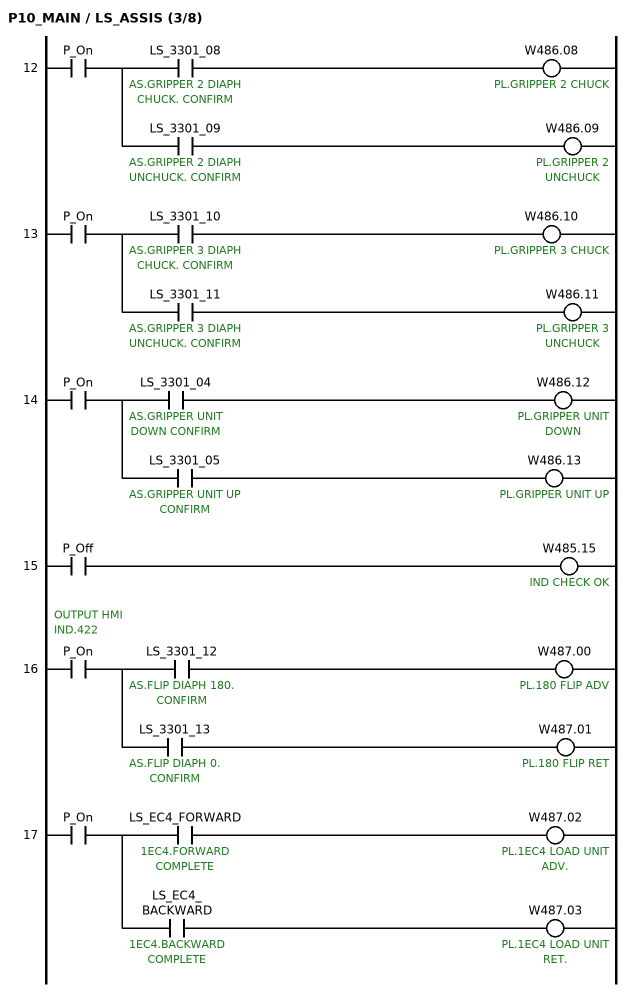
; [picture p48: P10_MAIN / LS_ASSIS, rungs 12-17]
; rung 12
LD P_On
OUT TR0
AND LS_3301_08  ; AS.GRIPPER 2 DIAPH CHUCK. CONFIRM
OUT W486.08  ; PL.GRIPPER 2 CHUCK
LD TR0
AND LS_3301_09  ; AS.GRIPPER 2 DIAPH UNCHUCK. CONFIRM
OUT W486.09  ; PL.GRIPPER 2 UNCHUCK
; rung 13
LD P_On
OUT TR0
AND LS_3301_10  ; AS.GRIPPER 3 DIAPH CHUCK. CONFIRM
OUT W486.10  ; PL.GRIPPER 3 CHUCK
LD TR0
AND LS_3301_11  ; AS.GRIPPER 3 DIAPH UNCHUCK. CONFIRM
OUT W486.11  ; PL.GRIPPER 3 UNCHUCK
; rung 14
LD P_On
OUT TR0
AND LS_3301_04  ; AS.GRIPPER UNIT DOWN CONFIRM
OUT W486.12  ; PL.GRIPPER UNIT DOWN
LD TR0
AND LS_3301_05  ; AS.GRIPPER UNIT UP CONFIRM
OUT W486.13  ; PL.GRIPPER UNIT UP
; rung 15
LD P_Off
OUT W485.15  ; IND CHECK OK
; rung 16: OUTPUT HMI / IND.422
LD P_On
OUT TR0
AND LS_3301_12  ; AS.FLIP DIAPH 180. CONFIRM
OUT W487.00  ; PL.180 FLIP ADV
LD TR0
AND LS_3301_13  ; AS.FLIP DIAPH 0. CONFIRM
OUT W487.01  ; PL.180 FLIP RET
; rung 17
LD P_On
OUT TR0
AND LS_EC4_FORWARD  ; 1EC4.FORWARD COMPLETE
OUT W487.02  ; PL.1EC4 LOAD UNIT ADV.
LD TR0
AND LS_EC4_BACKWARD  ; 1EC4.BACKWARD COMPLETE
OUT W487.03  ; PL.1EC4 LOAD UNIT RET.

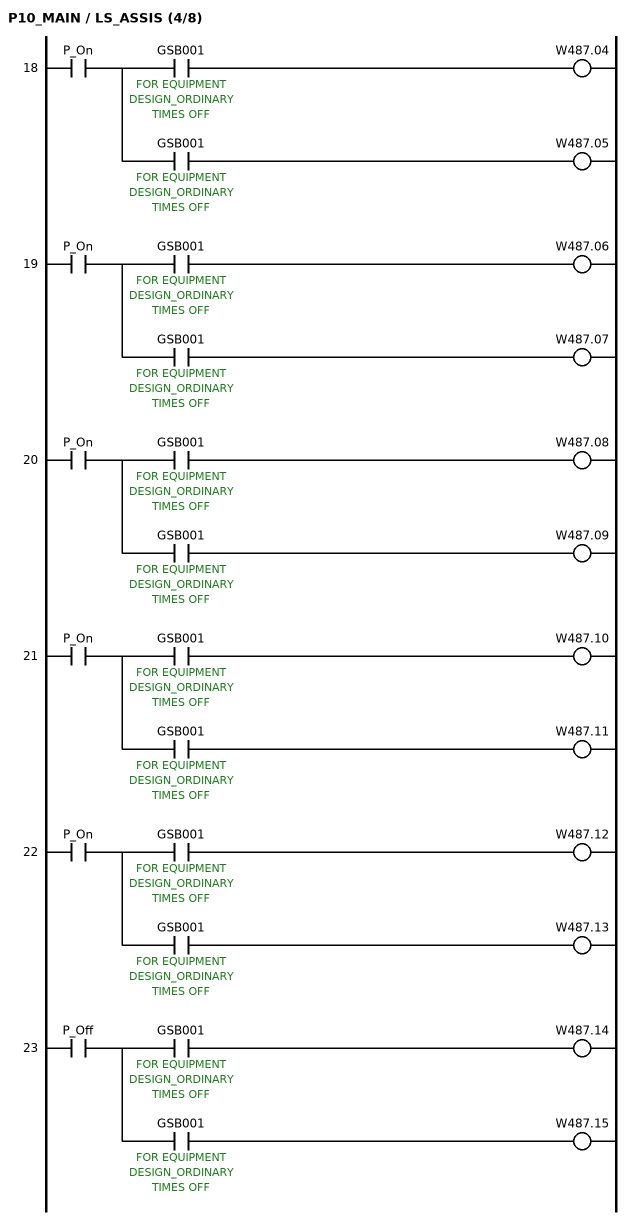
; rung 18
LD P_On
OUT TR0
AND GSB001  ; FOR EQUIPMENT DESIGN_ORDINARY TIMES OFF
OUT W487.04
LD TR0
AND GSB001  ; FOR EQUIPMENT DESIGN_ORDINARY TIMES OFF
OUT W487.05
; rung 19
LD P_On
OUT TR0
AND GSB001  ; FOR EQUIPMENT DESIGN_ORDINARY TIMES OFF
OUT W487.06
LD TR0
AND GSB001  ; FOR EQUIPMENT DESIGN_ORDINARY TIMES OFF
OUT W487.07
; rung 20
LD P_On
OUT TR0
AND GSB001  ; FOR EQUIPMENT DESIGN_ORDINARY TIMES OFF
OUT W487.08
LD TR0
AND GSB001  ; FOR EQUIPMENT DESIGN_ORDINARY TIMES OFF
OUT W487.09
; rung 21
LD P_On
OUT TR0
AND GSB001  ; FOR EQUIPMENT DESIGN_ORDINARY TIMES OFF
OUT W487.10
LD TR0
AND GSB001  ; FOR EQUIPMENT DESIGN_ORDINARY TIMES OFF
OUT W487.11
; rung 22
LD P_On
OUT TR0
AND GSB001  ; FOR EQUIPMENT DESIGN_ORDINARY TIMES OFF
OUT W487.12
LD TR0
AND GSB001  ; FOR EQUIPMENT DESIGN_ORDINARY TIMES OFF
OUT W487.13
; rung 23
LD P_Off
OUT TR0
AND GSB001  ; FOR EQUIPMENT DESIGN_ORDINARY TIMES OFF
OUT W487.14
LD TR0
AND GSB001  ; FOR EQUIPMENT DESIGN_ORDINARY TIMES OFF
OUT W487.15

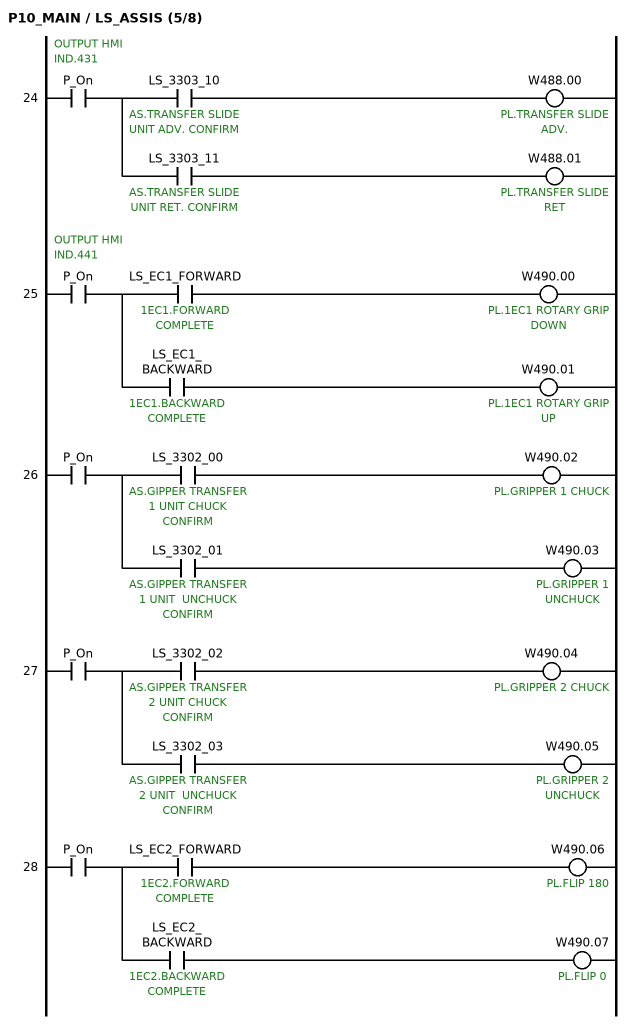
; rung 24: OUTPUT HMI / IND.431
LD P_On
OUT TR0
AND LS_3303_10  ; AS.TRANSFER SLIDE UNIT ADV. CONFIRM
OUT W488.00  ; PL.TRANSFER SLIDE ADV.
LD TR0
AND LS_3303_11  ; AS.TRANSFER SLIDE UNIT RET. CONFIRM
OUT W488.01  ; PL.TRANSFER SLIDE RET
; rung 25: OUTPUT HMI / IND.441
LD P_On
OUT TR0
AND LS_EC1_FORWARD  ; 1EC1.FORWARD COMPLETE
OUT W490.00  ; PL.1EC1 ROTARY GRIP DOWN
LD TR0
AND LS_EC1_BACKWARD  ; 1EC1.BACKWARD COMPLETE
OUT W490.01  ; PL.1EC1 ROTARY GRIP UP
; rung 26
LD P_On
OUT TR0
AND LS_3302_00  ; AS.GIPPER TRANSFER 1 UNIT CHUCK CONFIRM
OUT W490.02  ; PL.GRIPPER 1 CHUCK
LD TR0
AND LS_3302_01  ; AS.GIPPER TRANSFER 1 UNIT  UNCHUCK CONFIRM
OUT W490.03  ; PL.GRIPPER 1 UNCHUCK
; rung 27
LD P_On
OUT TR0
AND LS_3302_02  ; AS.GIPPER TRANSFER 2 UNIT CHUCK CONFIRM
OUT W490.04  ; PL.GRIPPER 2 CHUCK
LD TR0
AND LS_3302_03  ; AS.GIPPER TRANSFER 2 UNIT  UNCHUCK CONFIRM
OUT W490.05  ; PL.GRIPPER 2 UNCHUCK
; rung 28
LD P_On
OUT TR0
AND LS_EC2_FORWARD  ; 1EC2.FORWARD COMPLETE
OUT W490.06  ; PL.FLIP 180
LD TR0
AND LS_EC2_BACKWARD  ; 1EC2.BACKWARD COMPLETE
OUT W490.07  ; PL.FLIP 0

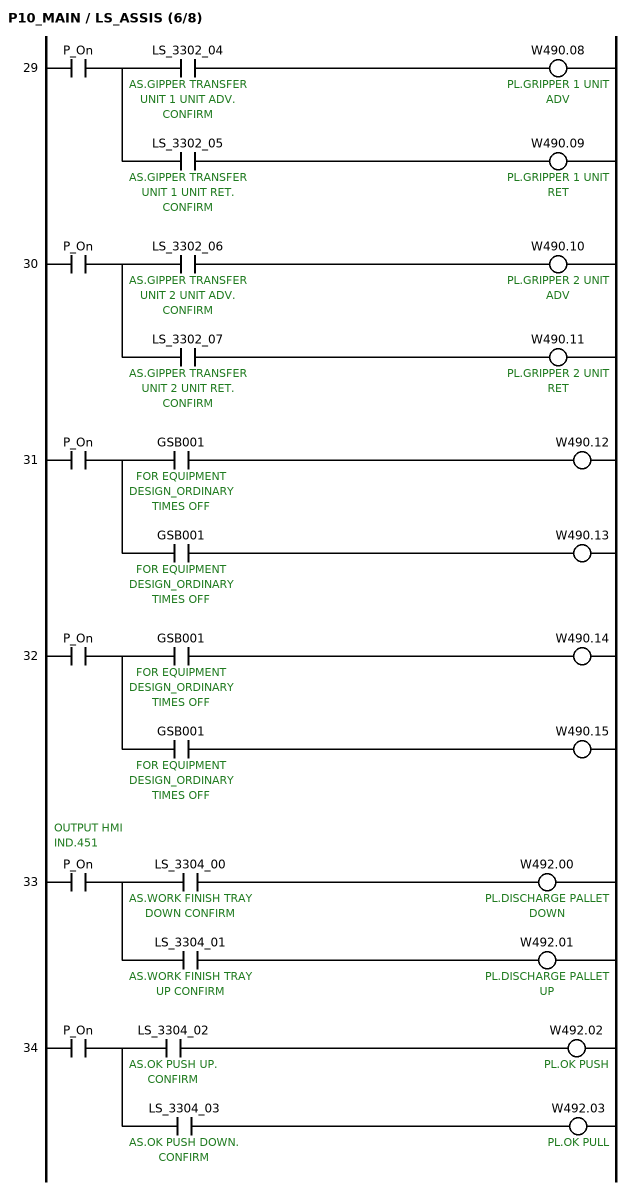
; rung 29
LD P_On
OUT TR0
AND LS_3302_04  ; AS.GIPPER TRANSFER UNIT 1 UNIT ADV. CONFIRM
OUT W490.08  ; PL.GRIPPER 1 UNIT ADV
LD TR0
AND LS_3302_05  ; AS.GIPPER TRANSFER UNIT 1 UNIT RET. CONFIRM
OUT W490.09  ; PL.GRIPPER 1 UNIT RET
; rung 30
LD P_On
OUT TR0
AND LS_3302_06  ; AS.GIPPER TRANSFER UNIT 2 UNIT ADV. CONFIRM
OUT W490.10  ; PL.GRIPPER 2 UNIT ADV
LD TR0
AND LS_3302_07  ; AS.GIPPER TRANSFER UNIT 2 UNIT RET. CONFIRM
OUT W490.11  ; PL.GRIPPER 2 UNIT RET
; rung 31
LD P_On
OUT TR0
AND GSB001  ; FOR EQUIPMENT DESIGN_ORDINARY TIMES OFF
OUT W490.12
LD TR0
AND GSB001  ; FOR EQUIPMENT DESIGN_ORDINARY TIMES OFF
OUT W490.13
; rung 32
LD P_On
OUT TR0
AND GSB001  ; FOR EQUIPMENT DESIGN_ORDINARY TIMES OFF
OUT W490.14
LD TR0
AND GSB001  ; FOR EQUIPMENT DESIGN_ORDINARY TIMES OFF
OUT W490.15
; rung 33: OUTPUT HMI / IND.451
LD P_On
OUT TR0
AND LS_3304_00  ; AS.WORK FINISH TRAY DOWN CONFIRM
OUT W492.00  ; PL.DISCHARGE PALLET DOWN
LD TR0
AND LS_3304_01  ; AS.WORK FINISH TRAY UP CONFIRM
OUT W492.01  ; PL.DISCHARGE PALLET UP
; rung 34
LD P_On
OUT TR0
AND LS_3304_02  ; AS.OK PUSH UP. CONFIRM
OUT W492.02  ; PL.OK PUSH
LD TR0
AND LS_3304_03  ; AS.OK PUSH DOWN. CONFIRM
OUT W492.03  ; PL.OK PULL

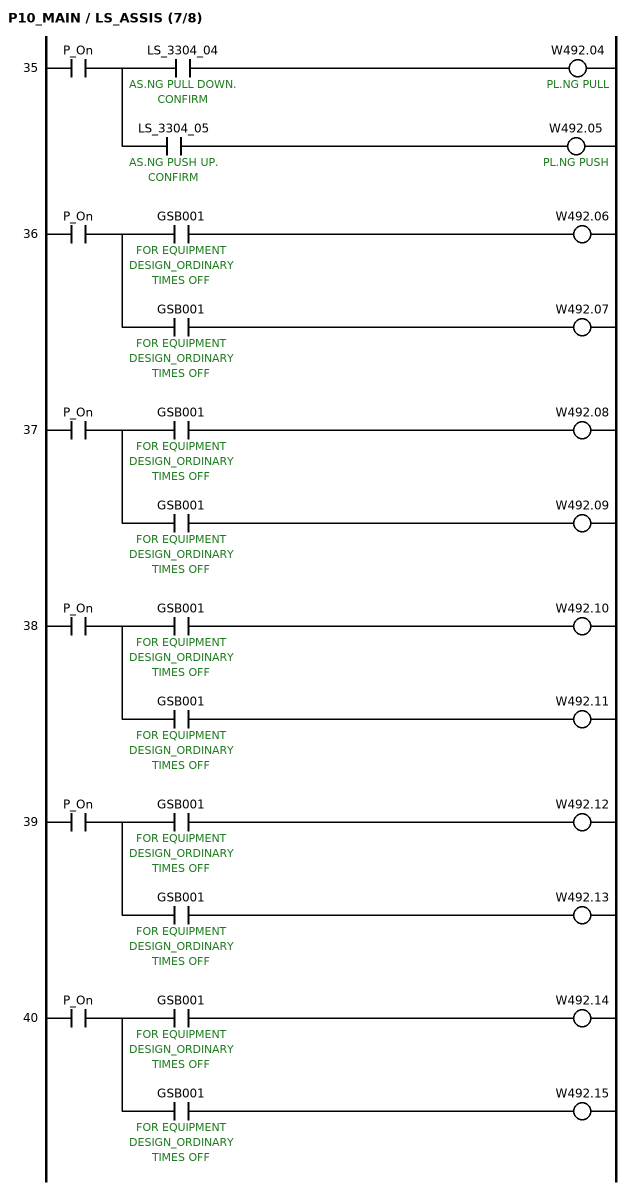
; rung 35
LD P_On
OUT TR0
AND LS_3304_04  ; AS.NG PULL DOWN. CONFIRM
OUT W492.04  ; PL.NG PULL
LD TR0
AND LS_3304_05  ; AS.NG PUSH UP. CONFIRM
OUT W492.05  ; PL.NG PUSH
; rung 36
LD P_On
OUT TR0
AND GSB001  ; FOR EQUIPMENT DESIGN_ORDINARY TIMES OFF
OUT W492.06
LD TR0
AND GSB001  ; FOR EQUIPMENT DESIGN_ORDINARY TIMES OFF
OUT W492.07
; rung 37
LD P_On
OUT TR0
AND GSB001  ; FOR EQUIPMENT DESIGN_ORDINARY TIMES OFF
OUT W492.08
LD TR0
AND GSB001  ; FOR EQUIPMENT DESIGN_ORDINARY TIMES OFF
OUT W492.09
; rung 38
LD P_On
OUT TR0
AND GSB001  ; FOR EQUIPMENT DESIGN_ORDINARY TIMES OFF
OUT W492.10
LD TR0
AND GSB001  ; FOR EQUIPMENT DESIGN_ORDINARY TIMES OFF
OUT W492.11
; rung 39
LD P_On
OUT TR0
AND GSB001  ; FOR EQUIPMENT DESIGN_ORDINARY TIMES OFF
OUT W492.12
LD TR0
AND GSB001  ; FOR EQUIPMENT DESIGN_ORDINARY TIMES OFF
OUT W492.13
; rung 40
LD P_On
OUT TR0
AND GSB001  ; FOR EQUIPMENT DESIGN_ORDINARY TIMES OFF
OUT W492.14
LD TR0
AND GSB001  ; FOR EQUIPMENT DESIGN_ORDINARY TIMES OFF
OUT W492.15

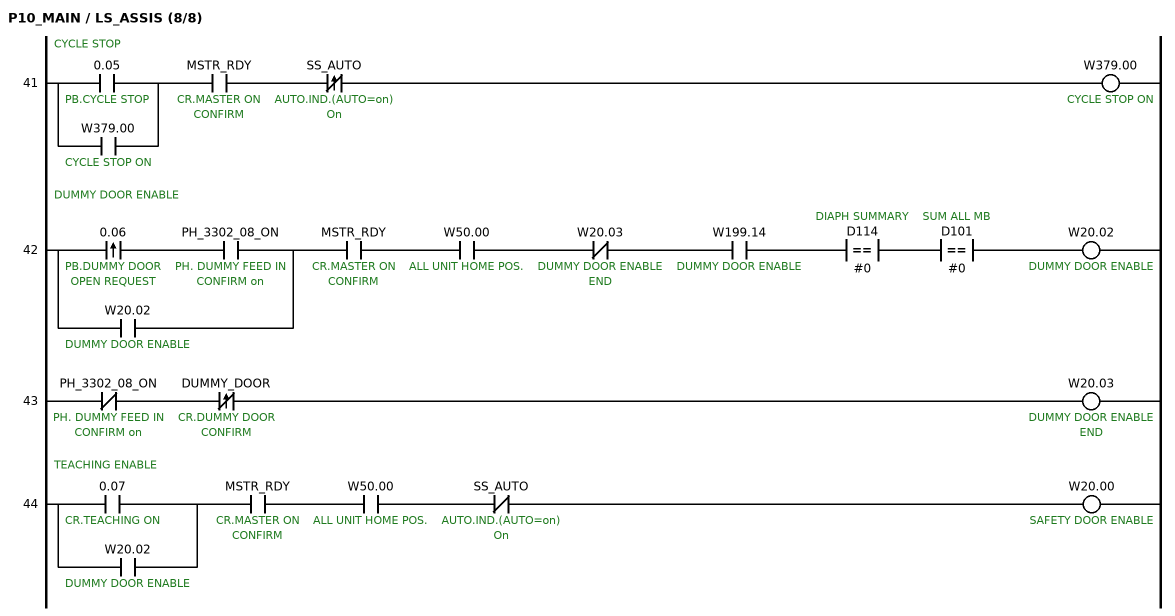
; rung 41: CYCLE STOP
LD 0.05  ; PB.CYCLE STOP
OR W379.00  ; CYCLE STOP ON
AND MSTR_RDY  ; CR.MASTER ON CONFIRM
@ANDNOT SS_AUTO  ; AUTO.IND.(AUTO=on) On
OUT W379.00  ; CYCLE STOP ON
; rung 42: DUMMY DOOR ENABLE
@LD 0.06  ; PB.DUMMY DOOR OPEN REQUEST
AND PH_3302_08_ON  ; PH. DUMMY FEED IN CONFIRM on
OR W20.02  ; DUMMY DOOR ENABLE
AND MSTR_RDY  ; CR.MASTER ON CONFIRM
AND W50.00  ; ALL UNIT HOME POS.
ANDNOT W20.03  ; DUMMY DOOR ENABLE END
AND W199.14  ; DUMMY DOOR ENABLE
AND=(300) D114 #0  ; DIAPH SUMMARY
AND=(300) D101 #0  ; SUM ALL MB
OUT W20.02  ; DUMMY DOOR ENABLE
; rung 43
LDNOT PH_3302_08_ON  ; PH. DUMMY FEED IN CONFIRM on
@ANDNOT DUMMY_DOOR  ; CR.DUMMY DOOR CONFIRM
OUT W20.03  ; DUMMY DOOR ENABLE END
; rung 44: TEACHING ENABLE
LD 0.07  ; CR.TEACHING ON
OR W20.02  ; DUMMY DOOR ENABLE
AND MSTR_RDY  ; CR.MASTER ON CONFIRM
AND W50.00  ; ALL UNIT HOME POS.
ANDNOT SS_AUTO  ; AUTO.IND.(AUTO=on) On
OUT W20.00  ; SAFETY DOOR ENABLE

### Section P08_MEMORY

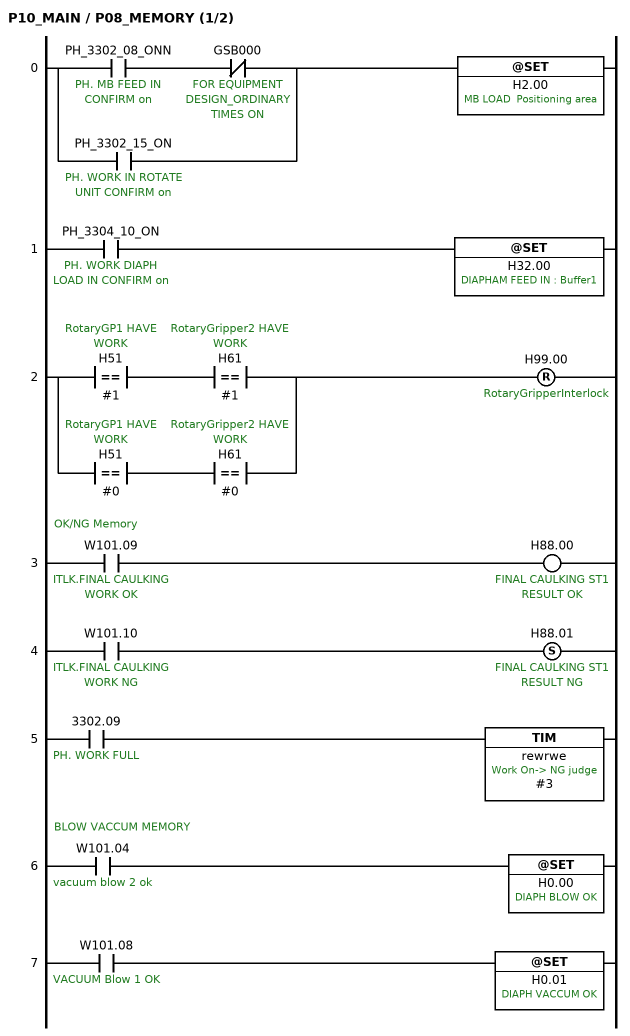
; rung 0
LD PH_3302_08_ONN  ; PH. MB FEED IN CONFIRM on
ANDNOT GSB000  ; FOR EQUIPMENT DESIGN_ORDINARY TIMES ON
OR PH_3302_15_ON  ; PH. WORK IN ROTATE UNIT CONFIRM on
@SET H2.00  ; MB LOAD  Positioning area
; rung 1
LD PH_3304_10_ON  ; PH. WORK DIAPH LOAD IN CONFIRM on
@SET H32.00  ; DIAPHAM FEED IN : Buffer1
; rung 2
LD=(300) H51 #1  ; RotaryGP1 HAVE WORK
AND=(300) H61 #1  ; RotaryGripper2 HAVE WORK
LD=(300) H51 #0  ; RotaryGP1 HAVE WORK
AND=(300) H61 #0  ; RotaryGripper2 HAVE WORK
ORLD
RSET H99.00  ; RotaryGripperInterlock
; rung 3: OK/NG Memory
LD W101.09  ; ITLK.FINAL CAULKING WORK OK
OUT H88.00  ; FINAL CAULKING ST1 RESULT OK
; rung 4
LD W101.10  ; ITLK.FINAL CAULKING WORK NG
SET H88.01  ; FINAL CAULKING ST1 RESULT NG
; rung 5
LD 3302.09  ; PH. WORK FULL
TIM rewrwe #3  ; Work On-> NG judge
; rung 6: BLOW VACCUM MEMORY
LD W101.04  ; vacuum blow 2 ok
@SET H0.00  ; DIAPH BLOW OK
; rung 7
LD W101.08  ; VACUUM Blow 1 OK
@SET H0.01  ; DIAPH VACCUM OK

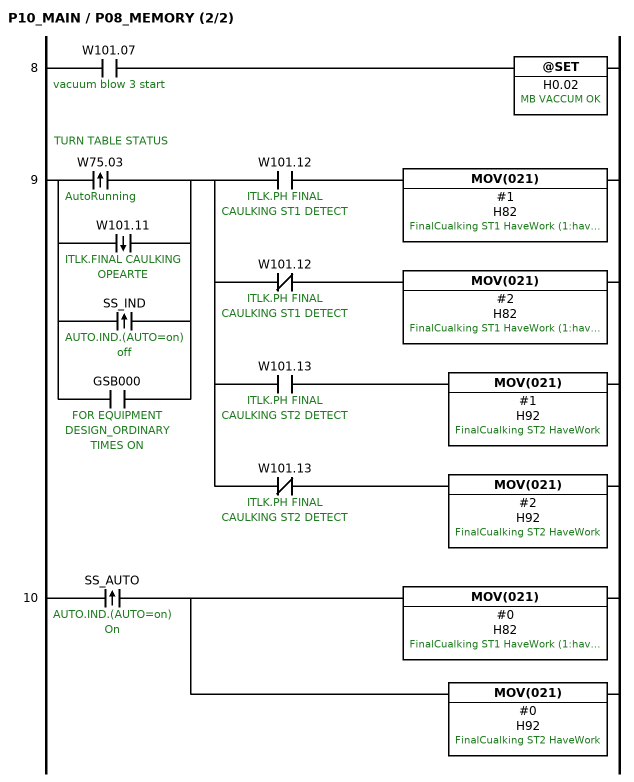
; rung 8
LD W101.07  ; vacuum blow 3 start
@SET H0.02  ; MB VACCUM OK
; rung 9: TURN TABLE STATUS
@LD W75.03  ; AutoRunning
%OR W101.11  ; ITLK.FINAL CAULKING OPEARTE
@OR SS_IND  ; AUTO.IND.(AUTO=on) off
OR GSB000  ; FOR EQUIPMENT DESIGN_ORDINARY TIMES ON
OUT TR0
AND W101.12  ; ITLK.PH FINAL CAULKING ST1 DETECT
MOV(021) #1 H82  ; FinalCualking ST1 HaveWork (1:have work 2:no work)
LD TR0
ANDNOT W101.12  ; ITLK.PH FINAL CAULKING ST1 DETECT
MOV(021) #2 H82  ; FinalCualking ST1 HaveWork (1:have work 2:no work)
LD TR0
AND W101.13  ; ITLK.PH FINAL CAULKING ST2 DETECT
MOV(021) #1 H92  ; FinalCualking ST2 HaveWork
LD TR0
ANDNOT W101.13  ; ITLK.PH FINAL CAULKING ST2 DETECT
MOV(021) #2 H92  ; FinalCualking ST2 HaveWork
; rung 10
@LD SS_AUTO  ; AUTO.IND.(AUTO=on) On
MOV(021) #0 H82  ; FinalCualking ST1 HaveWork (1:have work 2:no work)
MOV(021) #0 H92  ; FinalCualking ST2 HaveWork

### Section P09_CONDITION

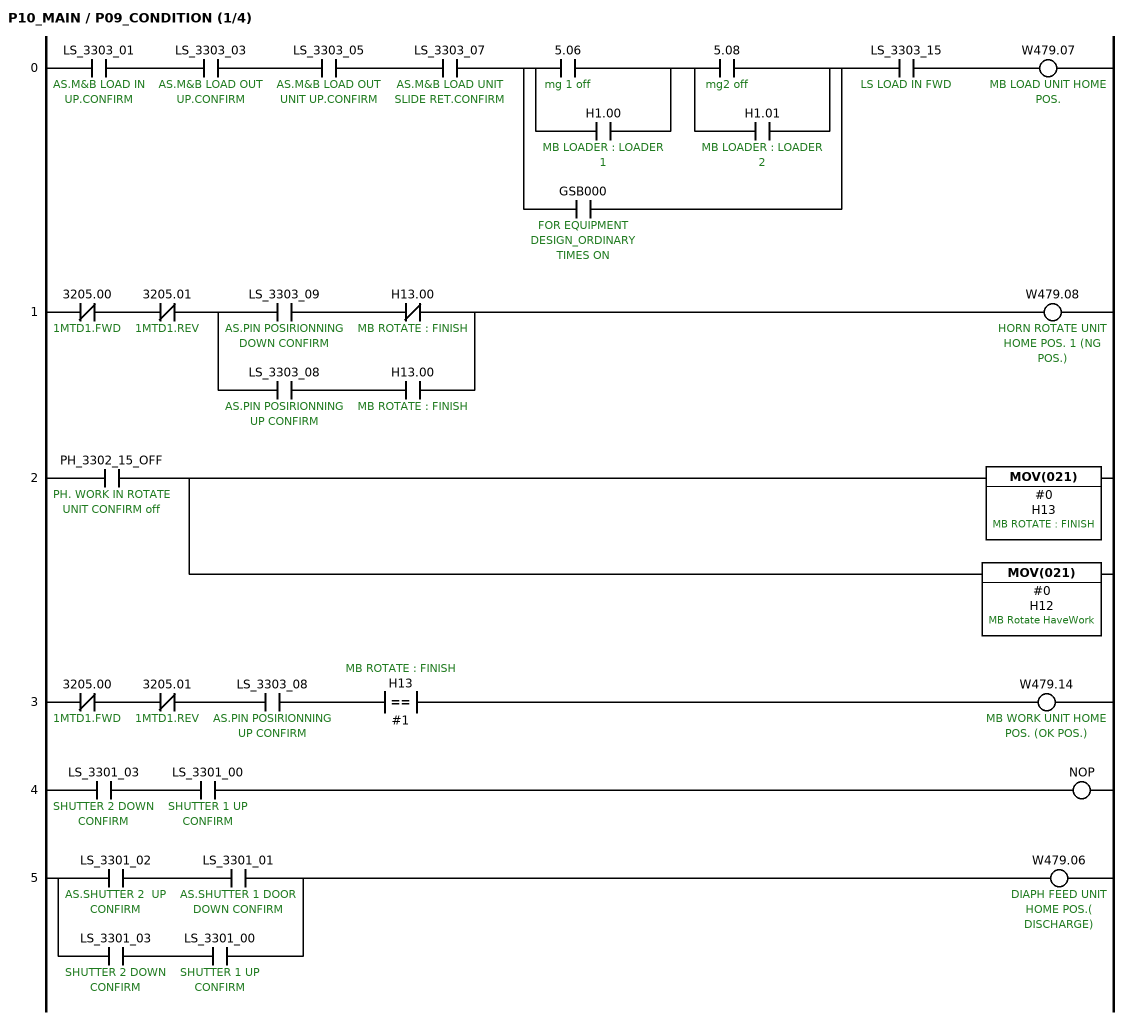
; rung 0
LD LS_3303_01  ; AS.M&B LOAD IN UP.CONFIRM
AND LS_3303_03  ; AS.M&B LOAD OUT UP.CONFIRM
AND LS_3303_05  ; AS.M&B LOAD OUT UNIT UP.CONFIRM
AND LS_3303_07  ; AS.M&B LOAD UNIT SLIDE RET.CONFIRM
LD 5.06  ; mg 1 off
OR H1.00  ; MB LOADER : LOADER 1
LD 5.08  ; mg2 off
OR H1.01  ; MB LOADER : LOADER 2
ANDLD
OR GSB000  ; FOR EQUIPMENT DESIGN_ORDINARY TIMES ON
ANDLD
AND LS_3303_15  ; LS LOAD IN FWD
OUT W479.07  ; MB LOAD UNIT HOME POS.
; rung 1
LDNOT 3205.00  ; 1MTD1.FWD
ANDNOT 3205.01  ; 1MTD1.REV
LD LS_3303_09  ; AS.PIN POSIRIONNING DOWN CONFIRM
ANDNOT H13.00  ; MB ROTATE : FINISH
LD LS_3303_08  ; AS.PIN POSIRIONNING UP CONFIRM
AND H13.00  ; MB ROTATE : FINISH
ORLD
ANDLD
OUT W479.08  ; HORN ROTATE UNIT HOME POS. 1 (NG POS.)
; rung 2
LD PH_3302_15_OFF  ; PH. WORK IN ROTATE UNIT CONFIRM off
MOV(021) #0 H13  ; MB ROTATE : FINISH
MOV(021) #0 H12  ; MB Rotate HaveWork
; rung 3
LDNOT 3205.00  ; 1MTD1.FWD
ANDNOT 3205.01  ; 1MTD1.REV
AND LS_3303_08  ; AS.PIN POSIRIONNING UP CONFIRM
AND=(300) H13 #1  ; MB ROTATE : FINISH
OUT W479.14  ; MB WORK UNIT HOME POS. (OK POS.)
; rung 4
LD LS_3301_03  ; SHUTTER 2 DOWN CONFIRM
AND LS_3301_00  ; SHUTTER 1 UP CONFIRM
OUT NOP
; rung 5
LD LS_3301_02  ; AS.SHUTTER 2  UP CONFIRM
AND LS_3301_01  ; AS.SHUTTER 1 DOOR DOWN CONFIRM
LD LS_3301_03  ; SHUTTER 2 DOWN CONFIRM
AND LS_3301_00  ; SHUTTER 1 UP CONFIRM
ORLD
OUT W479.06  ; DIAPH FEED UNIT HOME POS.(DISCHARGE)

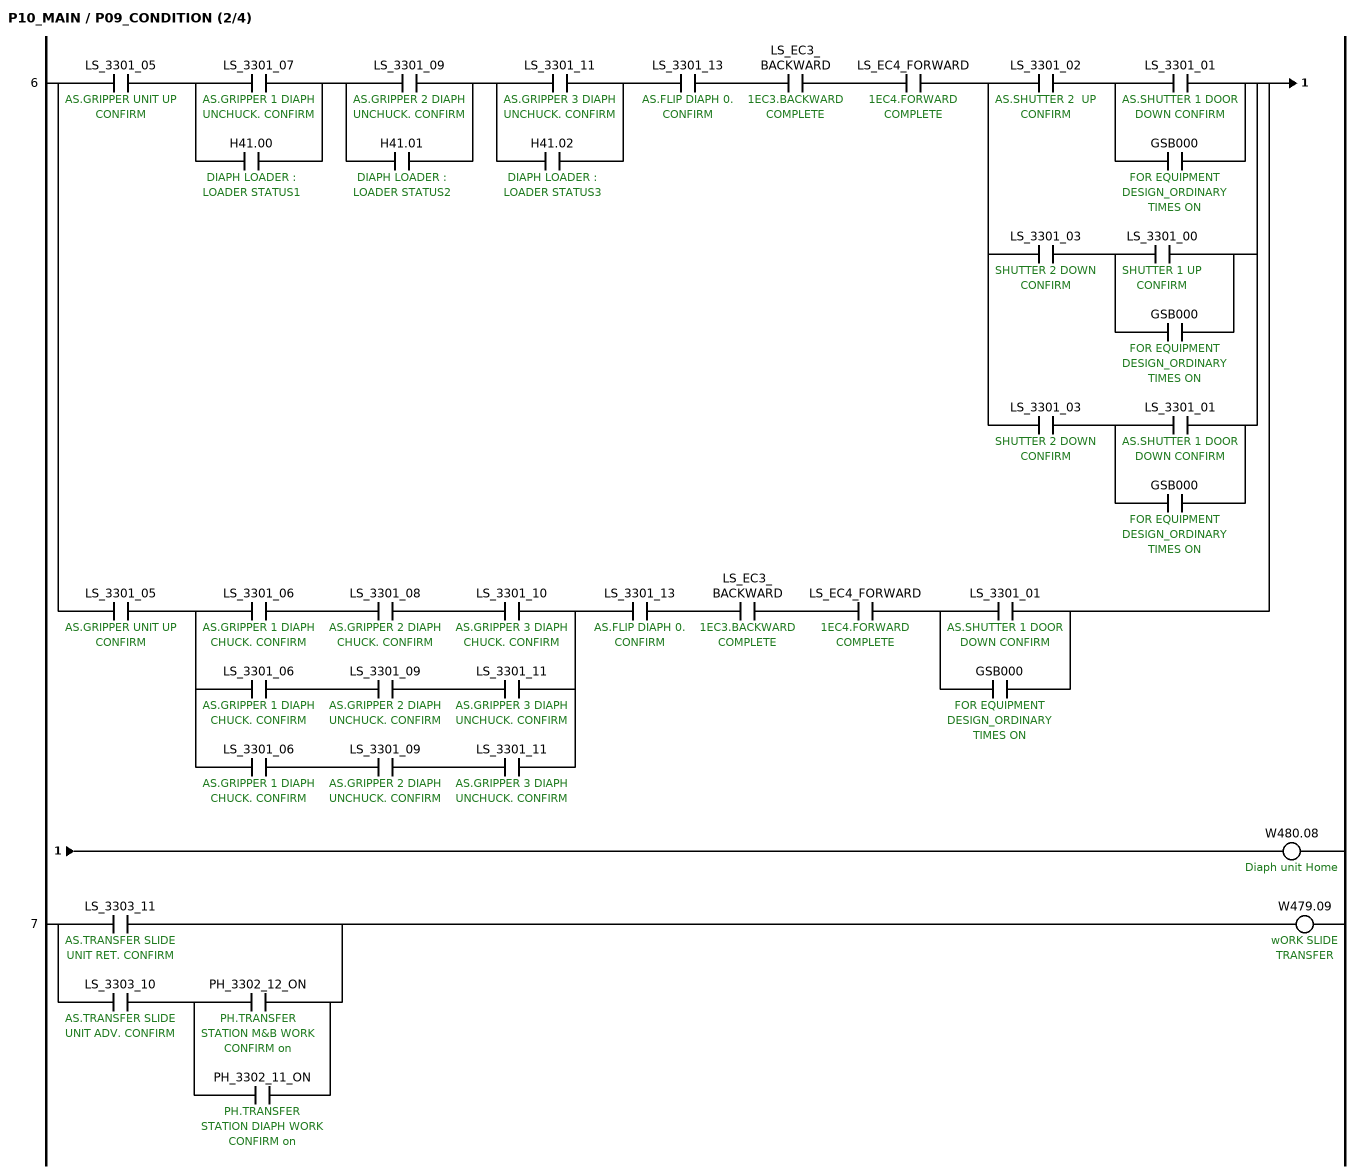
; rung 6
LD LS_3301_05  ; AS.GRIPPER UNIT UP CONFIRM
LD LS_3301_07  ; AS.GRIPPER 1 DIAPH UNCHUCK. CONFIRM
OR H41.00  ; DIAPH LOADER : LOADER STATUS1
ANDLD
LD LS_3301_09  ; AS.GRIPPER 2 DIAPH UNCHUCK. CONFIRM
OR H41.01  ; DIAPH LOADER : LOADER STATUS2
ANDLD
LD LS_3301_11  ; AS.GRIPPER 3 DIAPH UNCHUCK. CONFIRM
OR H41.02  ; DIAPH LOADER : LOADER STATUS3
ANDLD
AND LS_3301_13  ; AS.FLIP DIAPH 0. CONFIRM
AND LS_EC3_BACKWARD  ; 1EC3.BACKWARD COMPLETE
AND LS_EC4_FORWARD  ; 1EC4.FORWARD COMPLETE
LD LS_3301_02  ; AS.SHUTTER 2  UP CONFIRM
LD LS_3301_01  ; AS.SHUTTER 1 DOOR DOWN CONFIRM
OR GSB000  ; FOR EQUIPMENT DESIGN_ORDINARY TIMES ON
ANDLD
LD LS_3301_03  ; SHUTTER 2 DOWN CONFIRM
LD LS_3301_00  ; SHUTTER 1 UP CONFIRM
OR GSB000  ; FOR EQUIPMENT DESIGN_ORDINARY TIMES ON
ANDLD
ORLD
LD LS_3301_03  ; SHUTTER 2 DOWN CONFIRM
LD LS_3301_01  ; AS.SHUTTER 1 DOOR DOWN CONFIRM
OR GSB000  ; FOR EQUIPMENT DESIGN_ORDINARY TIMES ON
ANDLD
ORLD
ANDLD
LD LS_3301_05  ; AS.GRIPPER UNIT UP CONFIRM
LD LS_3301_06  ; AS.GRIPPER 1 DIAPH CHUCK. CONFIRM
AND LS_3301_08  ; AS.GRIPPER 2 DIAPH CHUCK. CONFIRM
AND LS_3301_10  ; AS.GRIPPER 3 DIAPH CHUCK. CONFIRM
LD LS_3301_06  ; AS.GRIPPER 1 DIAPH CHUCK. CONFIRM
AND LS_3301_09  ; AS.GRIPPER 2 DIAPH UNCHUCK. CONFIRM
AND LS_3301_11  ; AS.GRIPPER 3 DIAPH UNCHUCK. CONFIRM
ORLD
LD LS_3301_06  ; AS.GRIPPER 1 DIAPH CHUCK. CONFIRM
AND LS_3301_09  ; AS.GRIPPER 2 DIAPH UNCHUCK. CONFIRM
AND LS_3301_11  ; AS.GRIPPER 3 DIAPH UNCHUCK. CONFIRM
ORLD
ANDLD
AND LS_3301_13  ; AS.FLIP DIAPH 0. CONFIRM
AND LS_EC3_BACKWARD  ; 1EC3.BACKWARD COMPLETE
AND LS_EC4_FORWARD  ; 1EC4.FORWARD COMPLETE
LD LS_3301_01  ; AS.SHUTTER 1 DOOR DOWN CONFIRM
OR GSB000  ; FOR EQUIPMENT DESIGN_ORDINARY TIMES ON
ANDLD
ORLD
OUT W480.08  ; Diaph unit Home
; rung 7
LD LS_3303_11  ; AS.TRANSFER SLIDE UNIT RET. CONFIRM
LD LS_3303_10  ; AS.TRANSFER SLIDE UNIT ADV. CONFIRM
LD PH_3302_12_ON  ; PH.TRANSFER STATION M&B WORK CONFIRM on
OR PH_3302_11_ON  ; PH.TRANSFER STATION DIAPH WORK CONFIRM on
ANDLD
ORLD
OUT W479.09  ; wORK SLIDE TRANSFER

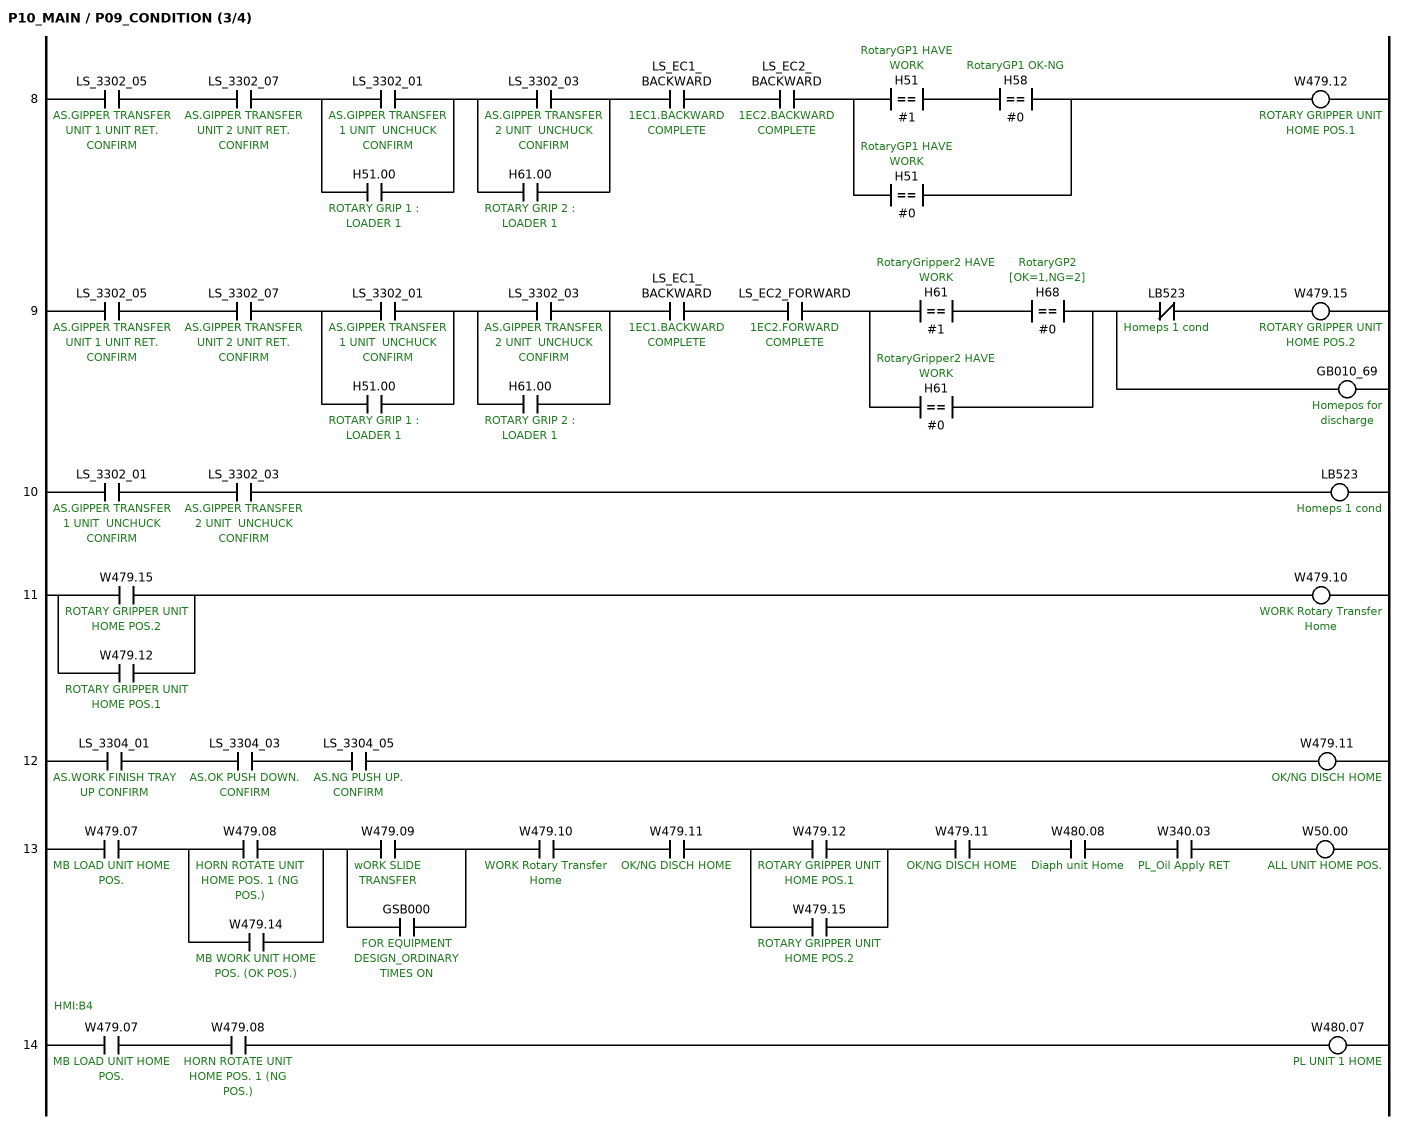
; rung 8
LD LS_3302_05  ; AS.GIPPER TRANSFER UNIT 1 UNIT RET. CONFIRM
AND LS_3302_07  ; AS.GIPPER TRANSFER UNIT 2 UNIT RET. CONFIRM
LD LS_3302_01  ; AS.GIPPER TRANSFER 1 UNIT  UNCHUCK CONFIRM
OR H51.00  ; ROTARY GRIP 1 : LOADER 1
ANDLD
LD LS_3302_03  ; AS.GIPPER TRANSFER 2 UNIT  UNCHUCK CONFIRM
OR H61.00  ; ROTARY GRIP 2 : LOADER 1
ANDLD
AND LS_EC1_BACKWARD  ; 1EC1.BACKWARD COMPLETE
AND LS_EC2_BACKWARD  ; 1EC2.BACKWARD COMPLETE
LD=(300) H51 #1  ; RotaryGP1 HAVE WORK
AND=(300) H58 #0  ; RotaryGP1 OK-NG
OR=(300) H51 #0  ; RotaryGP1 HAVE WORK
ANDLD
OUT W479.12  ; ROTARY GRIPPER UNIT HOME POS.1
; rung 9
LD LS_3302_05  ; AS.GIPPER TRANSFER UNIT 1 UNIT RET. CONFIRM
AND LS_3302_07  ; AS.GIPPER TRANSFER UNIT 2 UNIT RET. CONFIRM
LD LS_3302_01  ; AS.GIPPER TRANSFER 1 UNIT  UNCHUCK CONFIRM
OR H51.00  ; ROTARY GRIP 1 : LOADER 1
ANDLD
LD LS_3302_03  ; AS.GIPPER TRANSFER 2 UNIT  UNCHUCK CONFIRM
OR H61.00  ; ROTARY GRIP 2 : LOADER 1
ANDLD
AND LS_EC1_BACKWARD  ; 1EC1.BACKWARD COMPLETE
AND LS_EC2_FORWARD  ; 1EC2.FORWARD COMPLETE
LD=(300) H61 #1  ; RotaryGripper2 HAVE WORK
AND=(300) H68 #0  ; RotaryGP2 [OK=1,NG=2]
OR=(300) H61 #0  ; RotaryGripper2 HAVE WORK
ANDLD
OUT TR0
ANDNOT LB523  ; Homeps 1 cond
OUT W479.15  ; ROTARY GRIPPER UNIT HOME POS.2
LD TR0
OUT GB010_69  ; Homepos for discharge
; rung 10
LD LS_3302_01  ; AS.GIPPER TRANSFER 1 UNIT  UNCHUCK CONFIRM
AND LS_3302_03  ; AS.GIPPER TRANSFER 2 UNIT  UNCHUCK CONFIRM
OUT LB523  ; Homeps 1 cond
; rung 11
LD W479.15  ; ROTARY GRIPPER UNIT HOME POS.2
OR W479.12  ; ROTARY GRIPPER UNIT HOME POS.1
OUT W479.10  ; WORK Rotary Transfer Home
; rung 12
LD LS_3304_01  ; AS.WORK FINISH TRAY UP CONFIRM
AND LS_3304_03  ; AS.OK PUSH DOWN. CONFIRM
AND LS_3304_05  ; AS.NG PUSH UP. CONFIRM
OUT W479.11  ; OK/NG DISCH HOME
; rung 13
LD W479.07  ; MB LOAD UNIT HOME POS.
LD W479.08  ; HORN ROTATE UNIT HOME POS. 1 (NG POS.)
OR W479.14  ; MB WORK UNIT HOME POS. (OK POS.)
ANDLD
LD W479.09  ; wORK SLIDE TRANSFER
OR GSB000  ; FOR EQUIPMENT DESIGN_ORDINARY TIMES ON
ANDLD
AND W479.10  ; WORK Rotary Transfer Home
AND W479.11  ; OK/NG DISCH HOME
LD W479.12  ; ROTARY GRIPPER UNIT HOME POS.1
OR W479.15  ; ROTARY GRIPPER UNIT HOME POS.2
ANDLD
AND W479.11  ; OK/NG DISCH HOME
AND W480.08  ; Diaph unit Home
AND W340.03  ; PL_Oil Apply RET
OUT W50.00  ; ALL UNIT HOME POS.
; rung 14: HMI:B4
LD W479.07  ; MB LOAD UNIT HOME POS.
AND W479.08  ; HORN ROTATE UNIT HOME POS. 1 (NG POS.)
OUT W480.07  ; PL UNIT 1 HOME

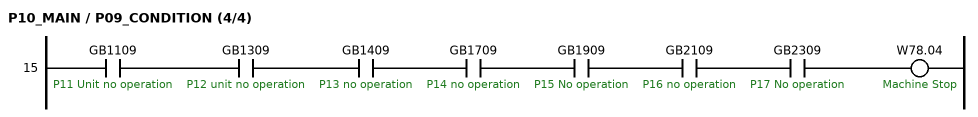
; rung 15
LD GB1109  ; P11 Unit no operation
AND GB1309  ; P12 unit no operation
AND GB1409  ; P13 no operation
AND GB1709  ; P14 no operation
AND GB1909  ; P15 No operation
AND GB2109  ; P16 no operation
AND GB2309  ; P17 No operation
OUT W78.04  ; Machine Stop

### Section P10_AUTO_MAIN

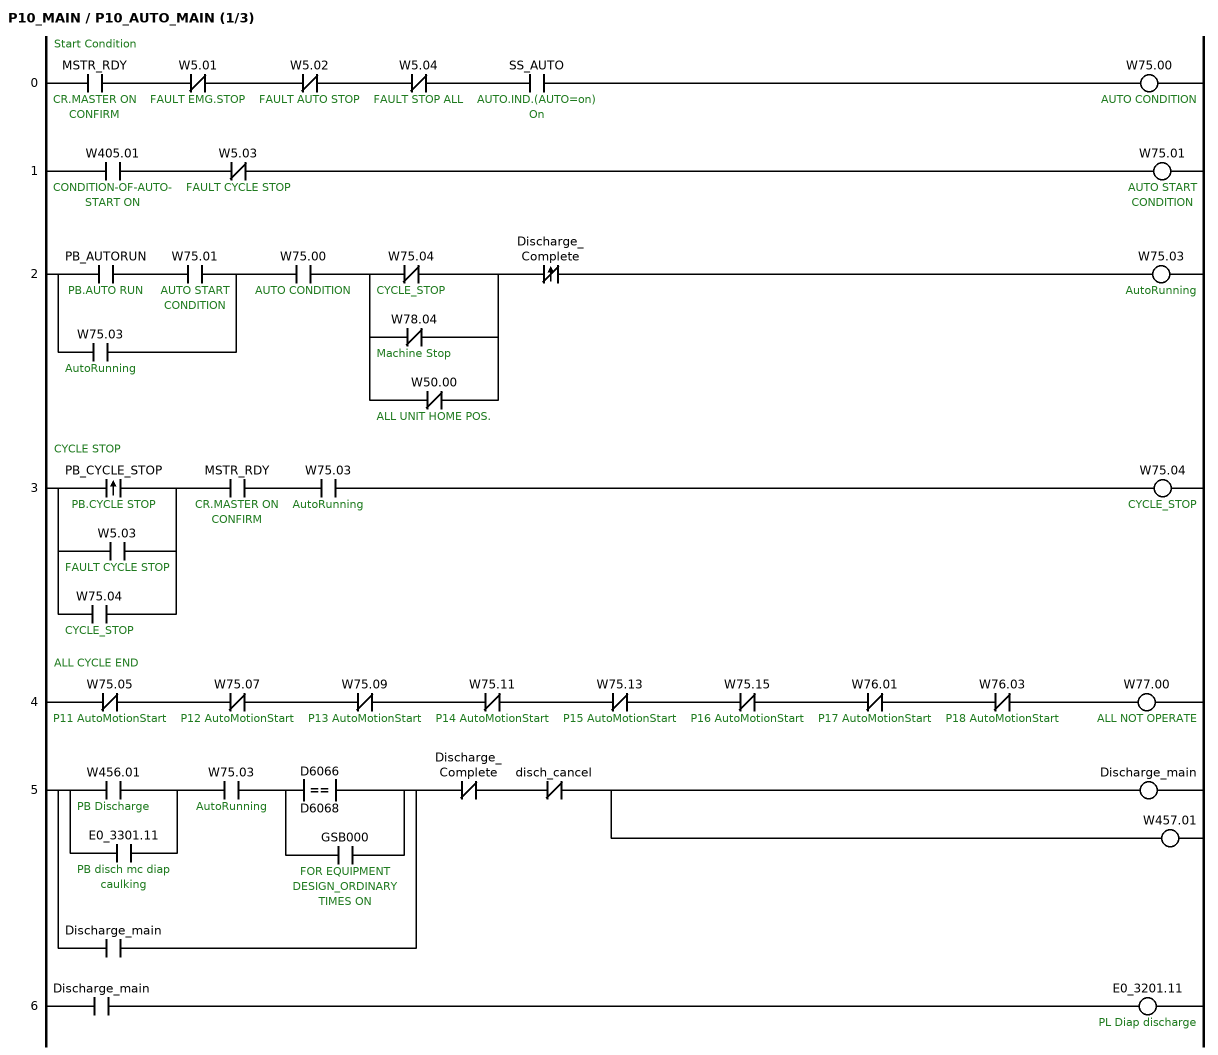
; rung 0: Start Condition
LD MSTR_RDY  ; CR.MASTER ON CONFIRM
ANDNOT W5.01  ; FAULT EMG.STOP
ANDNOT W5.02  ; FAULT AUTO STOP
ANDNOT W5.04  ; FAULT STOP ALL
AND SS_AUTO  ; AUTO.IND.(AUTO=on) On
OUT W75.00  ; AUTO CONDITION
; rung 1
LD W405.01  ; CONDITION-OF-AUTO-START ON
ANDNOT W5.03  ; FAULT CYCLE STOP
OUT W75.01  ; AUTO START CONDITION
; rung 2
LD PB_AUTORUN  ; PB.AUTO RUN
AND W75.01  ; AUTO START CONDITION
OR W75.03  ; AutoRunning
AND W75.00  ; AUTO CONDITION
LDNOT W75.04  ; CYCLE_STOP
ORNOT W78.04  ; Machine Stop
ORNOT W50.00  ; ALL UNIT HOME POS.
ANDLD
@ANDNOT Discharge_Complete
OUT W75.03  ; AutoRunning
; rung 3: CYCLE STOP
@LD PB_CYCLE_STOP  ; PB.CYCLE STOP
OR W5.03  ; FAULT CYCLE STOP
OR W75.04  ; CYCLE_STOP
AND MSTR_RDY  ; CR.MASTER ON CONFIRM
AND W75.03  ; AutoRunning
OUT W75.04  ; CYCLE_STOP
; rung 4: ALL CYCLE END
LDNOT W75.05  ; P11 AutoMotionStart
ANDNOT W75.07  ; P12 AutoMotionStart
ANDNOT W75.09  ; P13 AutoMotionStart
ANDNOT W75.11  ; P14 AutoMotionStart
ANDNOT W75.13  ; P15 AutoMotionStart
ANDNOT W75.15  ; P16 AutoMotionStart
ANDNOT W76.01  ; P17 AutoMotionStart
ANDNOT W76.03  ; P18 AutoMotionStart
OUT W77.00  ; ALL NOT OPERATE
; rung 5
LD W456.01  ; PB Discharge
OR E0_3301.11  ; PB disch mc diap caulking
AND W75.03  ; AutoRunning
LD=(300) D6066 D6068
OR GSB000  ; FOR EQUIPMENT DESIGN_ORDINARY TIMES ON
ANDLD
OR Discharge_main
ANDNOT Discharge_Complete
ANDNOT disch_cancel
OUT Discharge_main
OUT W457.01
; rung 6
LD Discharge_main
OUT E0_3201.11  ; PL Diap discharge

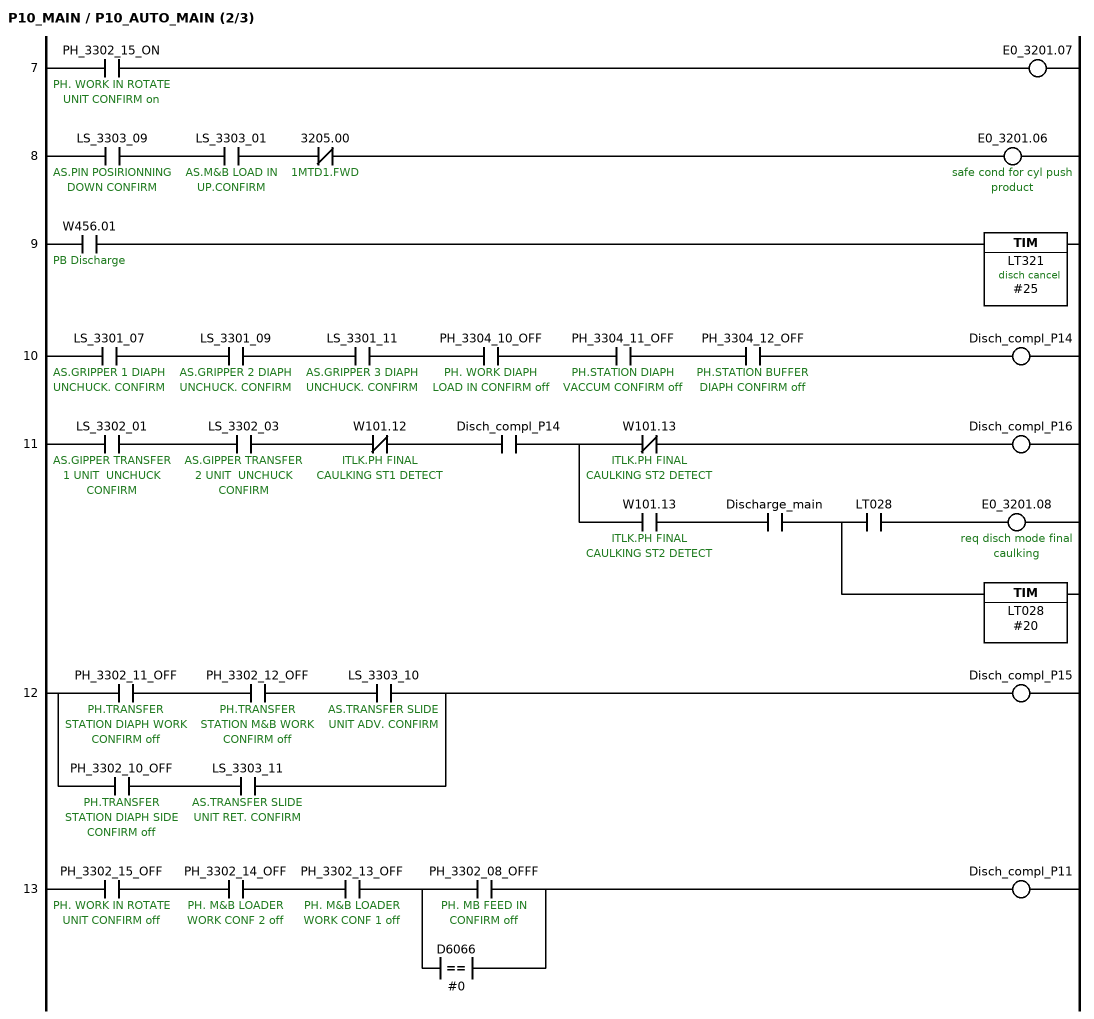
; rung 7
LD PH_3302_15_ON  ; PH. WORK IN ROTATE UNIT CONFIRM on
OUT E0_3201.07
; rung 8
LD LS_3303_09  ; AS.PIN POSIRIONNING DOWN CONFIRM
AND LS_3303_01  ; AS.M&B LOAD IN UP.CONFIRM
ANDNOT 3205.00  ; 1MTD1.FWD
OUT E0_3201.06  ; safe cond for cyl push product
; rung 9
LD W456.01  ; PB Discharge
TIM LT321 #25  ; disch cancel
; rung 10
LD LS_3301_07  ; AS.GRIPPER 1 DIAPH UNCHUCK. CONFIRM
AND LS_3301_09  ; AS.GRIPPER 2 DIAPH UNCHUCK. CONFIRM
AND LS_3301_11  ; AS.GRIPPER 3 DIAPH UNCHUCK. CONFIRM
AND PH_3304_10_OFF  ; PH. WORK DIAPH LOAD IN CONFIRM off
AND PH_3304_11_OFF  ; PH.STATION DIAPH VACCUM CONFIRM off
AND PH_3304_12_OFF  ; PH.STATION BUFFER DIAPH CONFIRM off
OUT Disch_compl_P14
; rung 11
LD LS_3302_01  ; AS.GIPPER TRANSFER 1 UNIT  UNCHUCK CONFIRM
AND LS_3302_03  ; AS.GIPPER TRANSFER 2 UNIT  UNCHUCK CONFIRM
ANDNOT W101.12  ; ITLK.PH FINAL CAULKING ST1 DETECT
AND Disch_compl_P14
OUT TR0
ANDNOT W101.13  ; ITLK.PH FINAL CAULKING ST2 DETECT
OUT Disch_compl_P16
LD TR0
AND W101.13  ; ITLK.PH FINAL CAULKING ST2 DETECT
AND Discharge_main
OUT TR0
AND LT028
OUT E0_3201.08  ; req disch mode final caulking
LD TR0
TIM LT028 #20
; rung 12
LD PH_3302_11_OFF  ; PH.TRANSFER STATION DIAPH WORK CONFIRM off
AND PH_3302_12_OFF  ; PH.TRANSFER STATION M&B WORK CONFIRM off
AND LS_3303_10  ; AS.TRANSFER SLIDE UNIT ADV. CONFIRM
LD PH_3302_10_OFF  ; PH.TRANSFER STATION DIAPH SIDE CONFIRM off
AND LS_3303_11  ; AS.TRANSFER SLIDE UNIT RET. CONFIRM
ORLD
OUT Disch_compl_P15
; rung 13
LD PH_3302_15_OFF  ; PH. WORK IN ROTATE UNIT CONFIRM off
AND PH_3302_14_OFF  ; PH. M&B LOADER WORK CONF 2 off
AND PH_3302_13_OFF  ; PH. M&B LOADER WORK CONF 1 off
LD PH_3302_08_OFFF  ; PH. MB FEED IN CONFIRM off
OR=(300) D6066 #0
ANDLD
OUT Disch_compl_P11

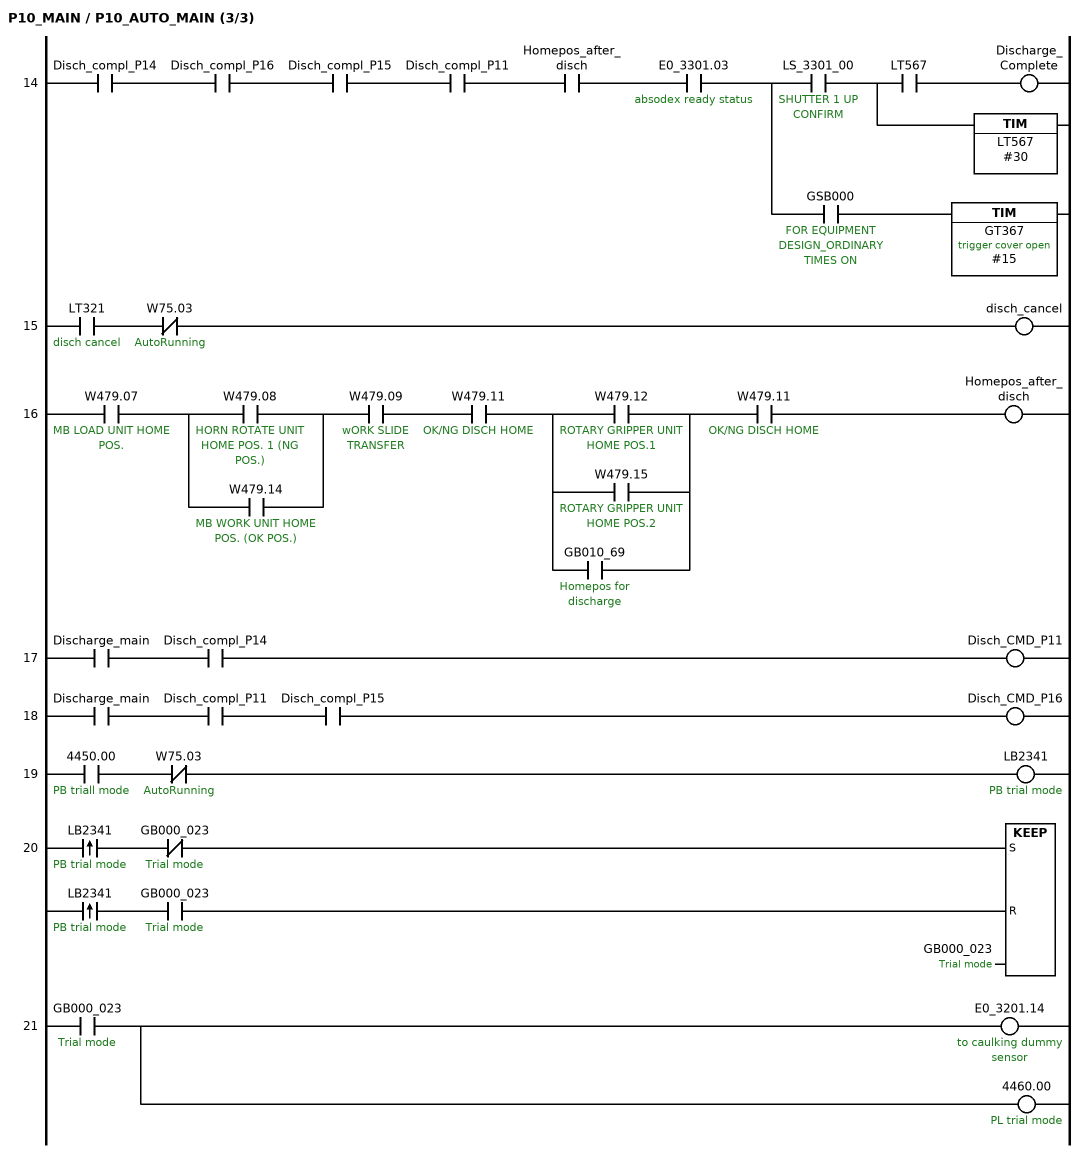
; rung 14
LD Disch_compl_P14
AND Disch_compl_P16
AND Disch_compl_P15
AND Disch_compl_P11
AND Homepos_after_disch
AND E0_3301.03  ; absodex ready status
OUT TR0
AND LS_3301_00  ; SHUTTER 1 UP CONFIRM
OUT TR1
AND LT567
OUT Discharge_Complete
LD TR1
TIM LT567 #30
LD TR0
AND GSB000  ; FOR EQUIPMENT DESIGN_ORDINARY TIMES ON
TIM GT367 #15  ; trigger cover open
; rung 15
LD LT321  ; disch cancel
ANDNOT W75.03  ; AutoRunning
OUT disch_cancel
; rung 16
LD W479.07  ; MB LOAD UNIT HOME POS.
LD W479.08  ; HORN ROTATE UNIT HOME POS. 1 (NG POS.)
OR W479.14  ; MB WORK UNIT HOME POS. (OK POS.)
ANDLD
AND W479.09  ; wORK SLIDE TRANSFER
AND W479.11  ; OK/NG DISCH HOME
LD W479.12  ; ROTARY GRIPPER UNIT HOME POS.1
OR W479.15  ; ROTARY GRIPPER UNIT HOME POS.2
OR GB010_69  ; Homepos for discharge
ANDLD
AND W479.11  ; OK/NG DISCH HOME
OUT Homepos_after_disch
; rung 17
LD Discharge_main
AND Disch_compl_P14
OUT Disch_CMD_P11
; rung 18
LD Discharge_main
AND Disch_compl_P11
AND Disch_compl_P15
OUT Disch_CMD_P16
; rung 19
LD 4450.00  ; PB triall mode
ANDNOT W75.03  ; AutoRunning
OUT LB2341  ; PB trial mode
; rung 20
@LD LB2341  ; PB trial mode
ANDNOT GB000_023  ; Trial mode
@LD LB2341  ; PB trial mode
AND GB000_023  ; Trial mode
KEEP GB000_023  ; Trial mode
; rung 21
LD GB000_023  ; Trial mode
OUT E0_3201.14  ; to caulking dummy sensor
OUT 4460.00  ; PL trial mode

### Section P20_WIP_CALCULATE

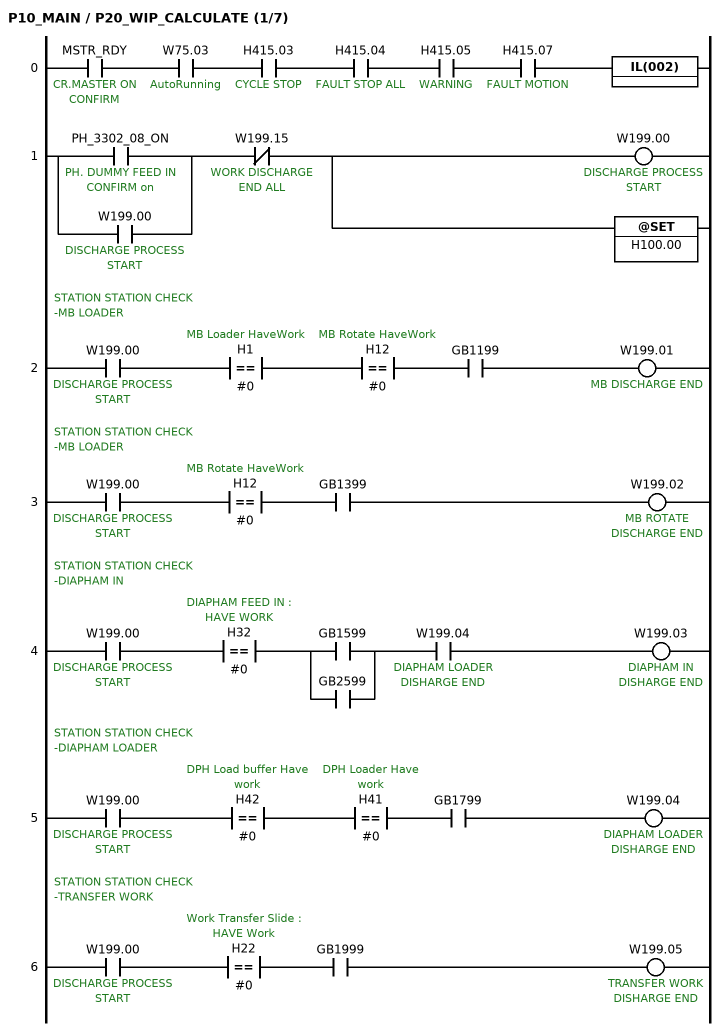
; rung 0
LD MSTR_RDY  ; CR.MASTER ON CONFIRM
AND W75.03  ; AutoRunning
AND H415.03  ; CYCLE STOP
AND H415.04  ; FAULT STOP ALL
AND H415.05  ; WARNING
AND H415.07  ; FAULT MOTION
IL(002)
; rung 1
LD PH_3302_08_ON  ; PH. DUMMY FEED IN CONFIRM on
OR W199.00  ; DISCHARGE PROCESS START
ANDNOT W199.15  ; WORK DISCHARGE END ALL
OUT W199.00  ; DISCHARGE PROCESS START
@SET H100.00
; rung 2: STATION STATION CHECK / -MB LOADER
LD W199.00  ; DISCHARGE PROCESS START
AND=(300) H1 #0  ; MB Loader HaveWork
AND=(300) H12 #0  ; MB Rotate HaveWork  // ROTATE UNIT NEED EMPTY
AND GB1199
OUT W199.01  ; MB DISCHARGE END
; rung 3: STATION STATION CHECK / -MB LOADER
LD W199.00  ; DISCHARGE PROCESS START
AND=(300) H12 #0  ; MB Rotate HaveWork
AND GB1399
OUT W199.02  ; MB ROTATE DISCHARGE END
; rung 4: STATION STATION CHECK / -DIAPHAM IN
LD W199.00  ; DISCHARGE PROCESS START
AND=(300) H32 #0  ; DIAPHAM FEED IN : HAVE WORK
LD GB1599
OR GB2599
ANDLD
AND W199.04  ; DIAPHAM LOADER DISHARGE END
OUT W199.03  ; DIAPHAM IN DISHARGE END
; rung 5: STATION STATION CHECK / -DIAPHAM LOADER
LD W199.00  ; DISCHARGE PROCESS START
AND=(300) H42 #0  ; DPH Load buffer Have work
AND=(300) H41 #0  ; DPH Loader Have work
AND GB1799
OUT W199.04  ; DIAPHAM LOADER DISHARGE END
; rung 6: STATION STATION CHECK / -TRANSFER WORK
LD W199.00  ; DISCHARGE PROCESS START
AND=(300) H22 #0  ; Work Transfer Slide : HAVE Work
AND GB1999
OUT W199.05  ; TRANSFER WORK DISHARGE END

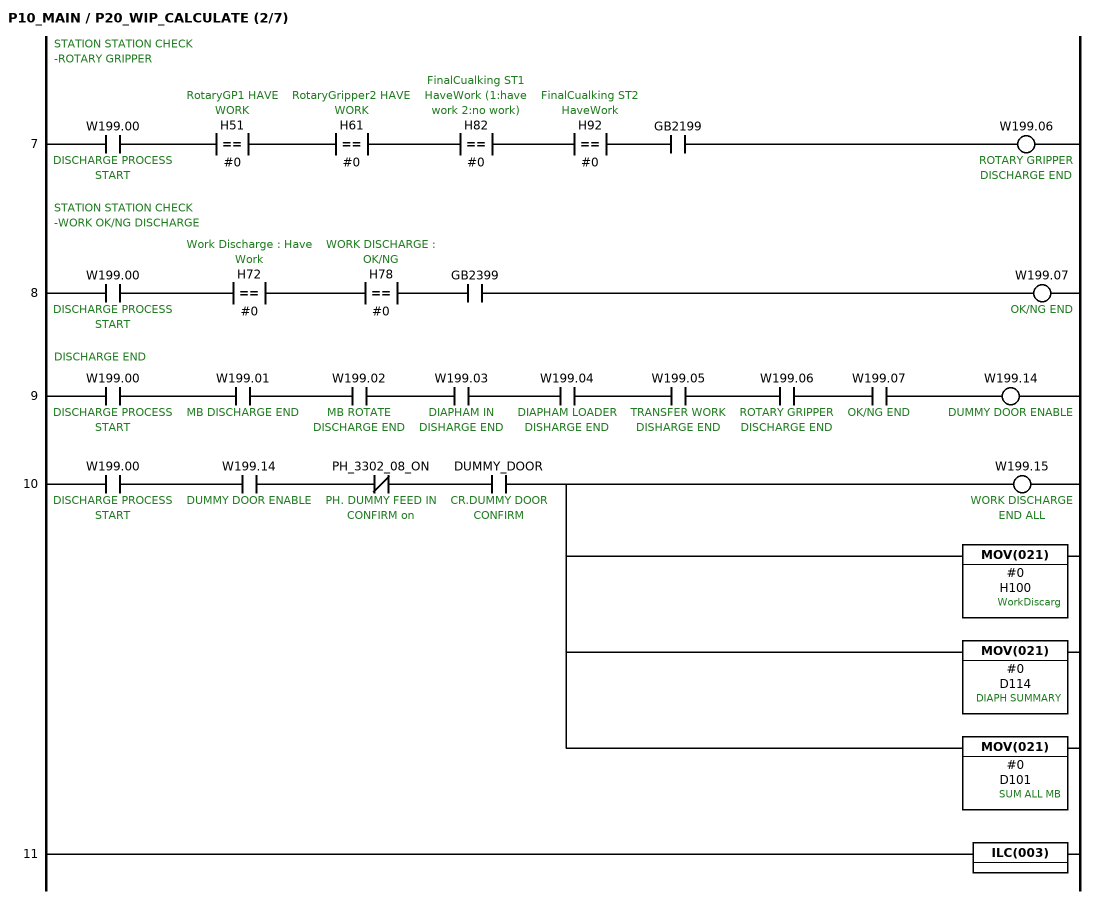
; rung 7: STATION STATION CHECK / -ROTARY GRIPPER
LD W199.00  ; DISCHARGE PROCESS START
AND=(300) H51 #0  ; RotaryGP1 HAVE WORK
AND=(300) H61 #0  ; RotaryGripper2 HAVE WORK
AND=(300) H82 #0  ; FinalCualking ST1 HaveWork (1:have work 2:no work)
AND=(300) H92 #0  ; FinalCualking ST2 HaveWork
AND GB2199
OUT W199.06  ; ROTARY GRIPPER DISCHARGE END
; rung 8: STATION STATION CHECK / -WORK OK/NG DISCHARGE
LD W199.00  ; DISCHARGE PROCESS START
AND=(300) H72 #0  ; Work Discharge : Have Work
AND=(300) H78 #0  ; WORK DISCHARGE : OK/NG
AND GB2399
OUT W199.07  ; OK/NG END
; rung 9: DISCHARGE END
LD W199.00  ; DISCHARGE PROCESS START
AND W199.01  ; MB DISCHARGE END
AND W199.02  ; MB ROTATE DISCHARGE END
AND W199.03  ; DIAPHAM IN DISHARGE END
AND W199.04  ; DIAPHAM LOADER DISHARGE END
AND W199.05  ; TRANSFER WORK DISHARGE END
AND W199.06  ; ROTARY GRIPPER DISCHARGE END
AND W199.07  ; OK/NG END
OUT W199.14  ; DUMMY DOOR ENABLE
; rung 10
LD W199.00  ; DISCHARGE PROCESS START
AND W199.14  ; DUMMY DOOR ENABLE
ANDNOT PH_3302_08_ON  ; PH. DUMMY FEED IN CONFIRM on
AND DUMMY_DOOR  ; CR.DUMMY DOOR CONFIRM
OUT W199.15  ; WORK DISCHARGE END ALL
MOV(021) #0 H100  ; WorkDiscarg
MOV(021) #0 D114  ; DIAPH SUMMARY
MOV(021) #0 D101  ; SUM ALL MB
; rung 11
ILC(003)

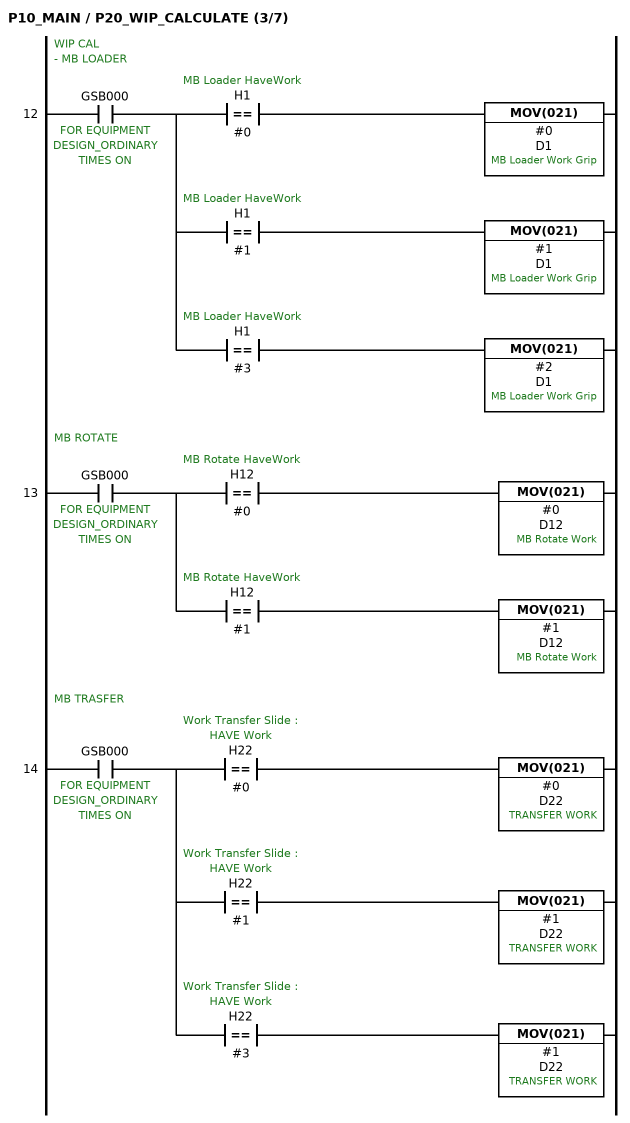
; rung 12: WIP CAL / - MB LOADER
LD GSB000  ; FOR EQUIPMENT DESIGN_ORDINARY TIMES ON
OUT TR0
AND=(300) H1 #0  ; MB Loader HaveWork
MOV(021) #0 D1  ; MB Loader Work Grip
LD TR0
AND=(300) H1 #1  ; MB Loader HaveWork
MOV(021) #1 D1  ; MB Loader Work Grip
LD TR0
AND=(300) H1 #3  ; MB Loader HaveWork
MOV(021) #2 D1  ; MB Loader Work Grip
; rung 13: MB ROTATE
LD GSB000  ; FOR EQUIPMENT DESIGN_ORDINARY TIMES ON
OUT TR0
AND=(300) H12 #0  ; MB Rotate HaveWork
MOV(021) #0 D12  ; MB Rotate Work
LD TR0
AND=(300) H12 #1  ; MB Rotate HaveWork
MOV(021) #1 D12  ; MB Rotate Work
; rung 14: MB TRASFER
LD GSB000  ; FOR EQUIPMENT DESIGN_ORDINARY TIMES ON
OUT TR0
AND=(300) H22 #0  ; Work Transfer Slide : HAVE Work
MOV(021) #0 D22  ; TRANSFER WORK
LD TR0
AND=(300) H22 #1  ; Work Transfer Slide : HAVE Work
MOV(021) #1 D22  ; TRANSFER WORK
LD TR0
AND=(300) H22 #3  ; Work Transfer Slide : HAVE Work
MOV(021) #1 D22  ; TRANSFER WORK

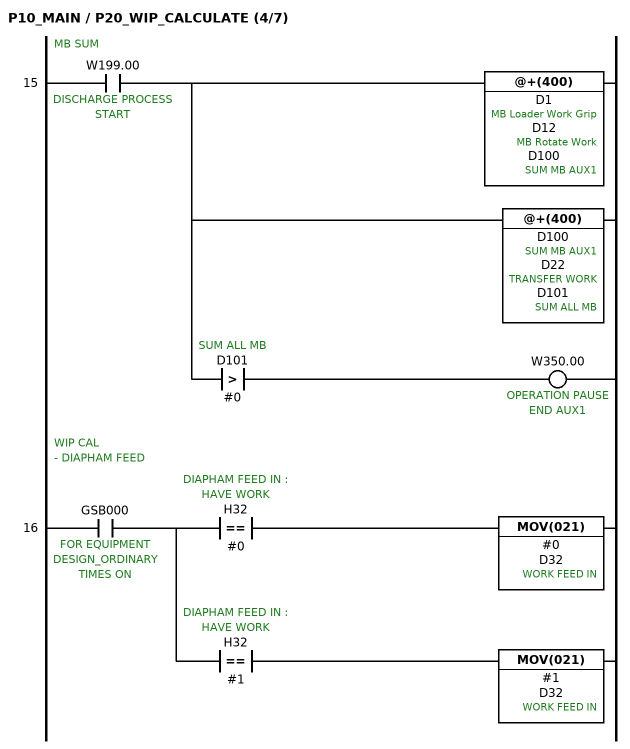
; rung 15: MB SUM
LD W199.00  ; DISCHARGE PROCESS START
@+(400) D1 D12 D100  ; MB Loader Work Grip, MB Rotate Work, SUM MB AUX1
@+(400) D100 D22 D101  ; SUM MB AUX1, TRANSFER WORK, SUM ALL MB
AND>(320) D101 #0  ; SUM ALL MB
OUT W350.00  ; OPERATION PAUSE END AUX1
; rung 16: WIP CAL / - DIAPHAM FEED
LD GSB000  ; FOR EQUIPMENT DESIGN_ORDINARY TIMES ON
OUT TR0
AND=(300) H32 #0  ; DIAPHAM FEED IN : HAVE WORK
MOV(021) #0 D32  ; WORK FEED IN
LD TR0
AND=(300) H32 #1  ; DIAPHAM FEED IN : HAVE WORK
MOV(021) #1 D32  ; WORK FEED IN

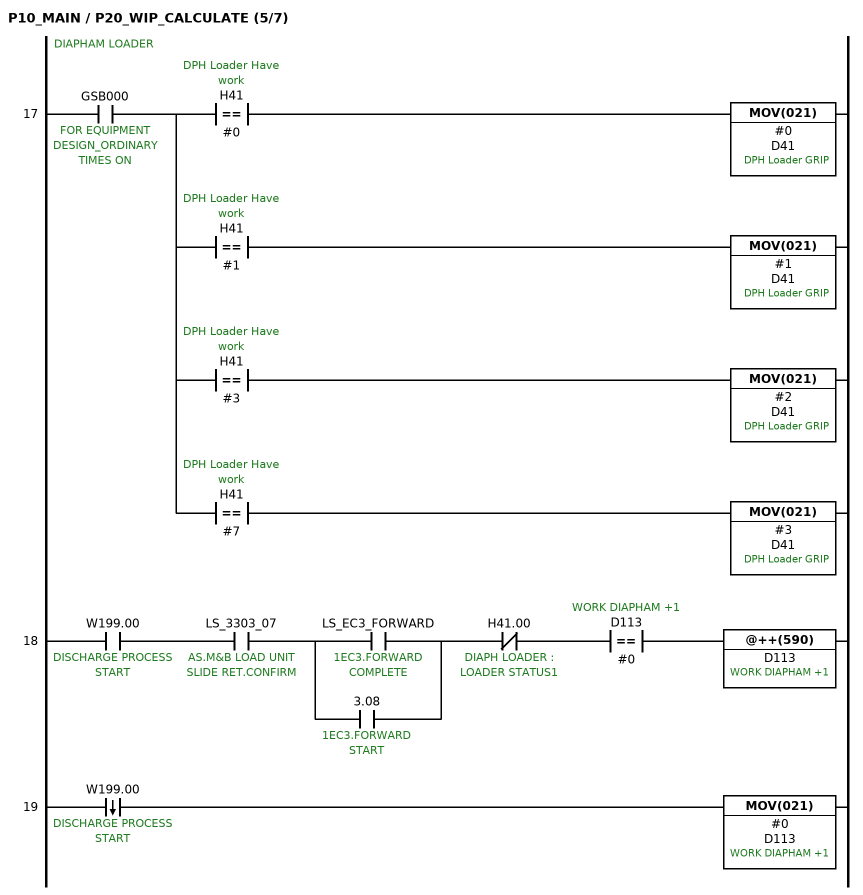
; rung 17: DIAPHAM LOADER
LD GSB000  ; FOR EQUIPMENT DESIGN_ORDINARY TIMES ON
OUT TR0
AND=(300) H41 #0  ; DPH Loader Have work
MOV(021) #0 D41  ; DPH Loader GRIP
LD TR0
AND=(300) H41 #1  ; DPH Loader Have work
MOV(021) #1 D41  ; DPH Loader GRIP
LD TR0
AND=(300) H41 #3  ; DPH Loader Have work
MOV(021) #2 D41  ; DPH Loader GRIP
LD TR0
AND=(300) H41 #7  ; DPH Loader Have work
MOV(021) #3 D41  ; DPH Loader GRIP
; rung 18
LD W199.00  ; DISCHARGE PROCESS START
AND LS_3303_07  ; AS.M&B LOAD UNIT SLIDE RET.CONFIRM
LD LS_EC3_FORWARD  ; 1EC3.FORWARD COMPLETE
OR 3.08  ; 1EC3.FORWARD START
ANDLD
ANDNOT H41.00  ; DIAPH LOADER : LOADER STATUS1
AND=(300) D113 #0  ; WORK DIAPHAM +1
@++(590) D113  ; WORK DIAPHAM +1
; rung 19
%LD W199.00  ; DISCHARGE PROCESS START
MOV(021) #0 D113  ; WORK DIAPHAM +1

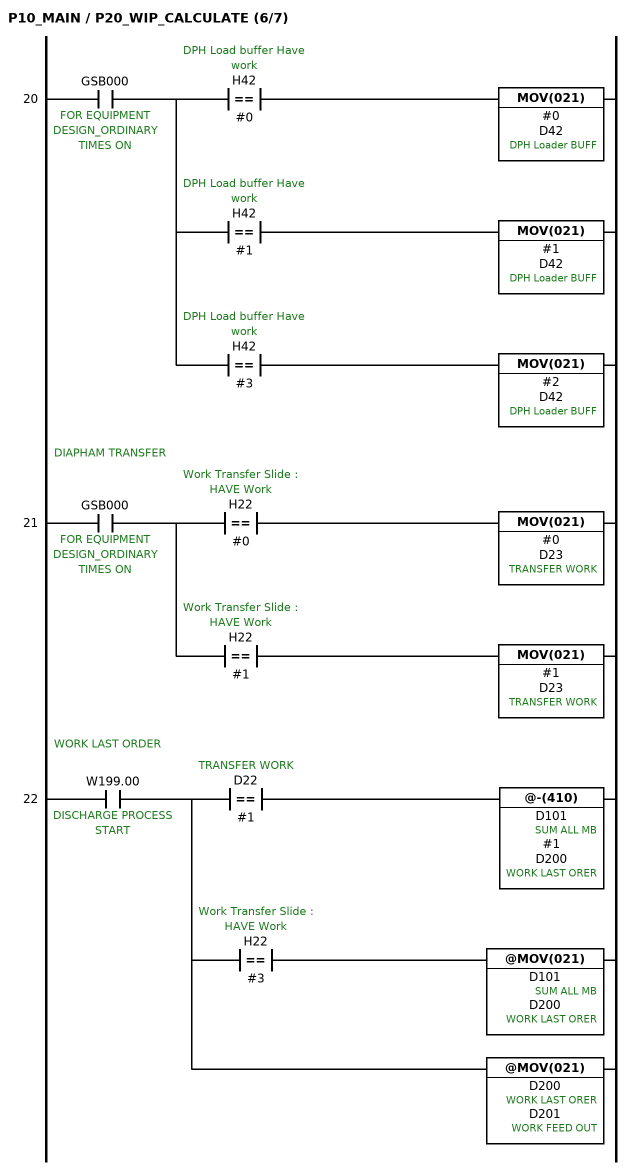
; rung 20
LD GSB000  ; FOR EQUIPMENT DESIGN_ORDINARY TIMES ON
OUT TR0
AND=(300) H42 #0  ; DPH Load buffer Have work
MOV(021) #0 D42  ; DPH Loader BUFF
LD TR0
AND=(300) H42 #1  ; DPH Load buffer Have work
MOV(021) #1 D42  ; DPH Loader BUFF
LD TR0
AND=(300) H42 #3  ; DPH Load buffer Have work
MOV(021) #2 D42  ; DPH Loader BUFF
; rung 21: DIAPHAM TRANSFER
LD GSB000  ; FOR EQUIPMENT DESIGN_ORDINARY TIMES ON
OUT TR0
AND=(300) H22 #0  ; Work Transfer Slide : HAVE Work
MOV(021) #0 D23  ; TRANSFER WORK
LD TR0
AND=(300) H22 #1  ; Work Transfer Slide : HAVE Work
MOV(021) #1 D23  ; TRANSFER WORK
; rung 22: WORK LAST ORDER
LD W199.00  ; DISCHARGE PROCESS START
OUT TR0
AND=(300) D22 #1  ; TRANSFER WORK
@-(410) D101 #1 D200  ; SUM ALL MB, WORK LAST ORER
LD TR0
AND=(300) H22 #3  ; Work Transfer Slide : HAVE Work
@MOV(021) D101 D200  ; SUM ALL MB, WORK LAST ORER
LD TR0
@MOV(021) D200 D201  ; WORK LAST ORER, WORK FEED OUT

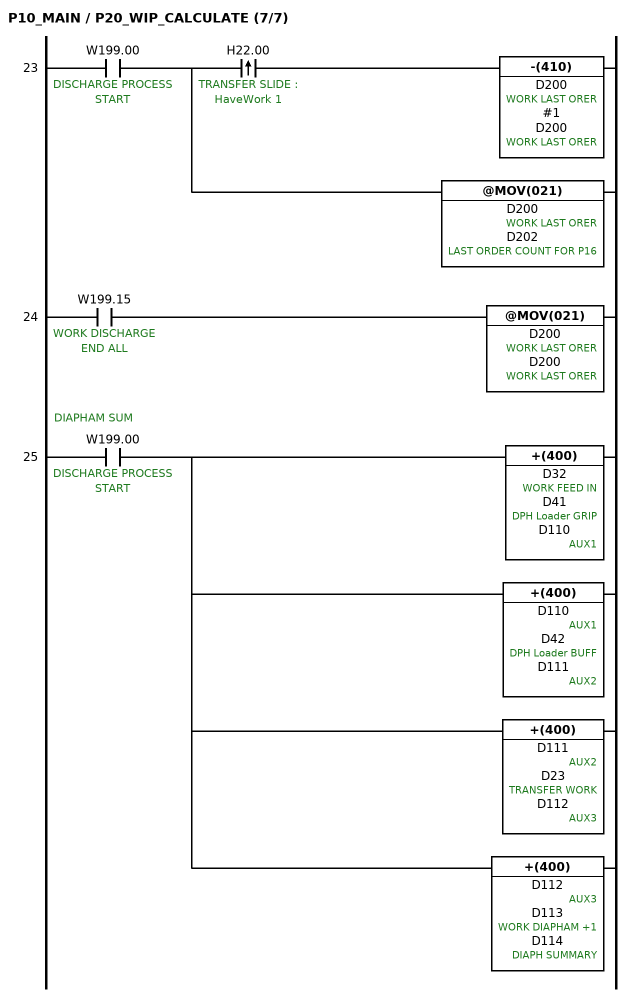
; rung 23
LD W199.00  ; DISCHARGE PROCESS START
OUT TR0
@AND H22.00  ; TRANSFER SLIDE : HaveWork 1
-(410) D200 #1 D200  ; WORK LAST ORER
LD TR0
@MOV(021) D200 D202  ; WORK LAST ORER, LAST ORDER COUNT FOR P16
; rung 24
LD W199.15  ; WORK DISCHARGE END ALL
@MOV(021) D200 D200  ; WORK LAST ORER
; rung 25: DIAPHAM SUM
LD W199.00  ; DISCHARGE PROCESS START
+(400) D32 D41 D110  ; WORK FEED IN, DPH Loader GRIP, AUX1
+(400) D110 D42 D111  ; AUX1, DPH Loader BUFF, AUX2
+(400) D111 D23 D112  ; AUX2, TRANSFER WORK, AUX3
+(400) D112 D113 D114  ; AUX3, WORK DIAPHAM +1, DIAPH SUMMARY

### Section COUNTER_MODEL

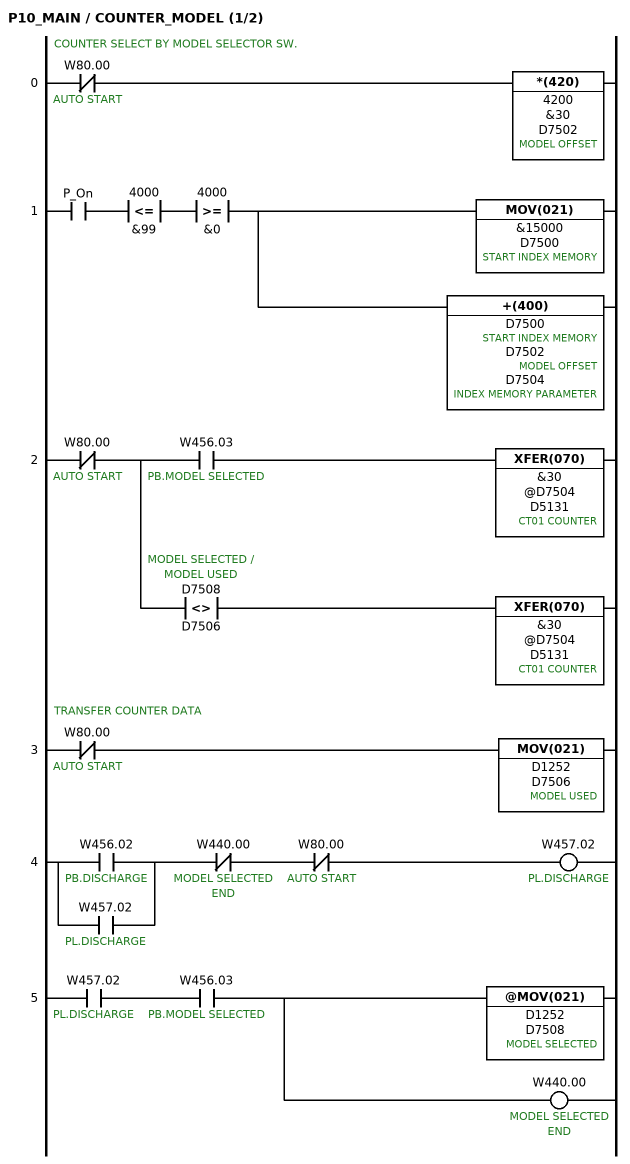
; rung 0: COUNTER SELECT BY MODEL SELECTOR SW.
LDNOT W80.00  ; AUTO START
*(420) 4200 &30 D7502  ; MODEL OFFSET
; rung 1
LD P_On
AND<=(315) 4000 &99
AND>=(325) 4000 &0
MOV(021) &15000 D7500  ; START INDEX MEMORY
+(400) D7500 D7502 D7504  ; START INDEX MEMORY, MODEL OFFSET, INDEX MEMORY PARAMETER
; rung 2
LDNOT W80.00  ; AUTO START
OUT TR0
AND W456.03  ; PB.MODEL SELECTED
XFER(070) &30 @D7504 D5131  ; CT01 COUNTER
LD TR0
AND<>(305) D7508 D7506  ; MODEL SELECTED, MODEL USED
XFER(070) &30 @D7504 D5131  ; CT01 COUNTER
; rung 3: TRANSFER COUNTER DATA
LDNOT W80.00  ; AUTO START
MOV(021) D1252 D7506  ; MODEL USED
; rung 4
LD W456.02  ; PB.DISCHARGE
OR W457.02  ; PL.DISCHARGE
ANDNOT W440.00  ; MODEL SELECTED END
ANDNOT W80.00  ; AUTO START
OUT W457.02  ; PL.DISCHARGE
; rung 5
LD W457.02  ; PL.DISCHARGE
AND W456.03  ; PB.MODEL SELECTED
@MOV(021) D1252 D7508  ; MODEL SELECTED
OUT W440.00  ; MODEL SELECTED END

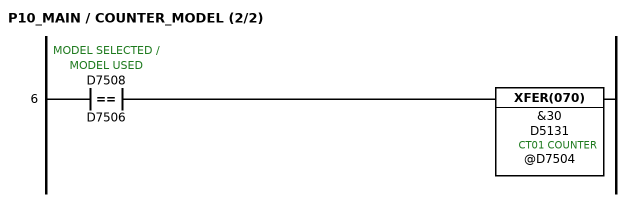
; rung 6
LD=(300) D7508 D7506  ; MODEL SELECTED, MODEL USED
XFER(070) &30 D5131 @D7504  ; CT01 COUNTER

### Section PB_SUB_V41

